% RSLogix 500 project I2P-Hands On 4 - Duncan_Sutton.RSS, saved by version 10.00.00.00 %
PROJECT "UNTITLED"    % processor: Bul.1763 MicroLogix 1100 Series B %

PROGRAM FILES
  LAD 2   15 rungs

DATA FILES
  O0 OUTPUT  4 elements
  I1 INPUT  6 elements
  S2 STATUS  66 elements
  B3 BINARY  1 elements
  T4 TIMER  1 elements
  C5 COUNTER  1 elements
  R6 CONTROL  1 elements
  N7 INTEGER  1 elements
  F8 FLOAT  1 elements

LADDER 2
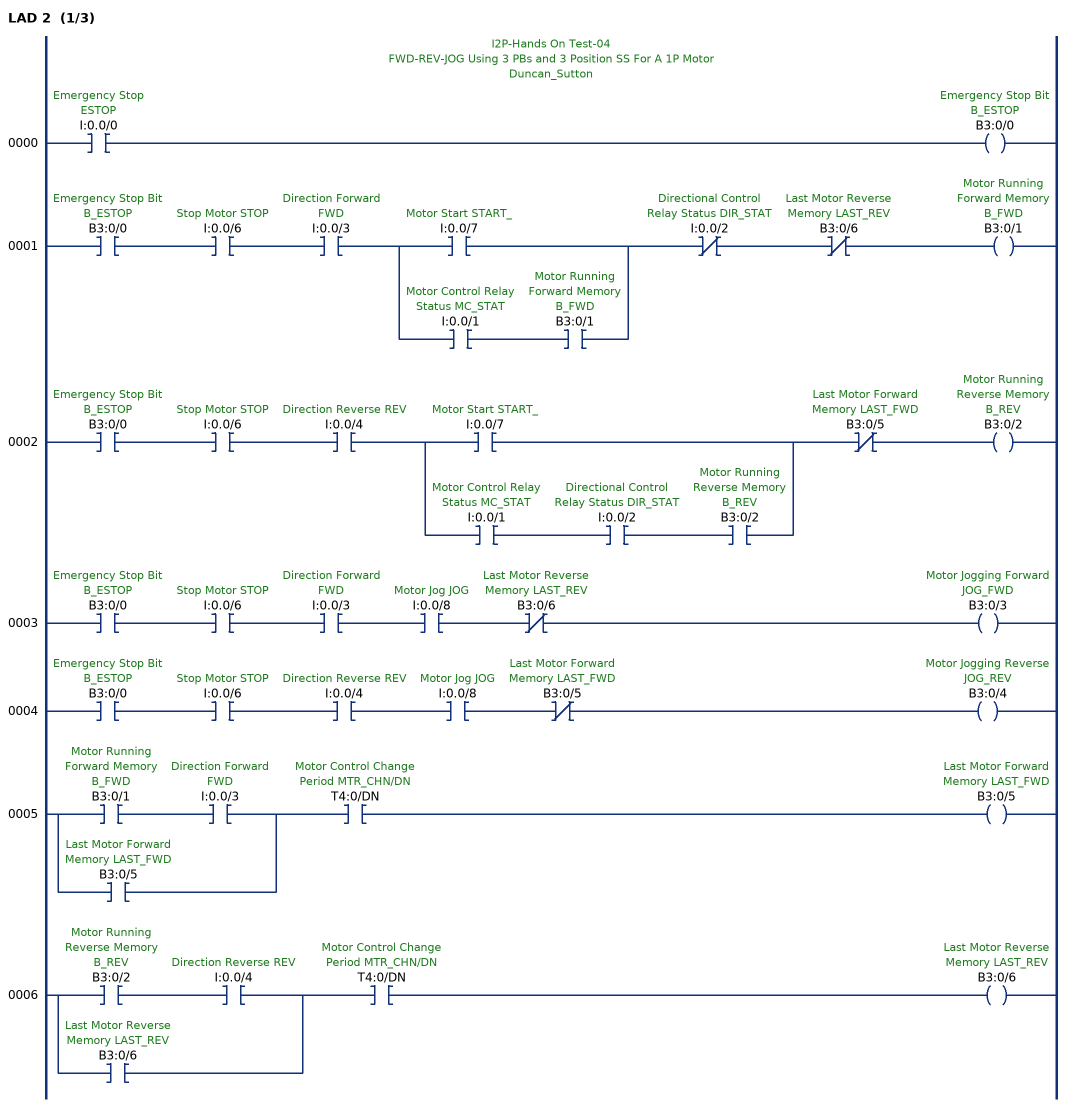
% Rung: 0 %
% I2P-Hands On Test-04
% FWD-REV-JOG Using 3 PBs and 3 Position SS For A 1P Motor
% Duncan_Sutton %
SOR XIC I:0.0/0 OTE B3:0/0 EOR
%   I:0.0/0  ESTOP  "Emergency Stop" %
%   B3:0/0  B_ESTOP  "Emergency Stop Bit" %
% Rung: 1 %
SOR XIC B3:0/0 XIC I:0.0/6 XIC I:0.0/3 BST XIC I:0.0/7 NXB XIC I:0.0/1 XIC B3:0/1 BND XIO I:0.0/2 XIO B3:0/6 OTE B3:0/1 EOR
%   B3:0/0  B_ESTOP  "Emergency Stop Bit" %
%   I:0.0/6  STOP  "Stop Motor" %
%   I:0.0/3  FWD  "Direction Forward" %
%   I:0.0/7  START_  "Motor Start" %
%   I:0.0/1  MC_STAT  "Motor Control Relay Status" %
%   B3:0/1  B_FWD  "Motor Running Forward Memory" %
%   I:0.0/2  DIR_STAT  "Directional Control Relay Status" %
%   B3:0/6  LAST_REV  "Last Motor Reverse Memory" %
% Rung: 2 %
SOR XIC B3:0/0 XIC I:0.0/6 XIC I:0.0/4 BST XIC I:0.0/7 NXB XIC I:0.0/1 XIC I:0.0/2 XIC B3:0/2 BND XIO B3:0/5 OTE B3:0/2 EOR
%   B3:0/0  B_ESTOP  "Emergency Stop Bit" %
%   I:0.0/6  STOP  "Stop Motor" %
%   I:0.0/4  REV  "Direction Reverse" %
%   I:0.0/7  START_  "Motor Start" %
%   I:0.0/1  MC_STAT  "Motor Control Relay Status" %
%   I:0.0/2  DIR_STAT  "Directional Control Relay Status" %
%   B3:0/2  B_REV  "Motor Running Reverse Memory" %
%   B3:0/5  LAST_FWD  "Last Motor Forward Memory" %
% Rung: 3 %
SOR XIC B3:0/0 XIC I:0.0/6 XIC I:0.0/3 XIC I:0.0/8 XIO B3:0/6 OTE B3:0/3 EOR
%   B3:0/0  B_ESTOP  "Emergency Stop Bit" %
%   I:0.0/6  STOP  "Stop Motor" %
%   I:0.0/3  FWD  "Direction Forward" %
%   I:0.0/8  JOG  "Motor Jog" %
%   B3:0/6  LAST_REV  "Last Motor Reverse Memory" %
%   B3:0/3  JOG_FWD  "Motor Jogging Forward" %
% Rung: 4 %
SOR XIC B3:0/0 XIC I:0.0/6 XIC I:0.0/4 XIC I:0.0/8 XIO B3:0/5 OTE B3:0/4 EOR
%   B3:0/0  B_ESTOP  "Emergency Stop Bit" %
%   I:0.0/6  STOP  "Stop Motor" %
%   I:0.0/4  REV  "Direction Reverse" %
%   I:0.0/8  JOG  "Motor Jog" %
%   B3:0/5  LAST_FWD  "Last Motor Forward Memory" %
%   B3:0/4  JOG_REV  "Motor Jogging Reverse" %
% Rung: 5 %
SOR BST XIC B3:0/1 XIC I:0.0/3 NXB XIC B3:0/5 BND XIC T4:0/DN OTE B3:0/5 EOR
%   B3:0/1  B_FWD  "Motor Running Forward Memory" %
%   I:0.0/3  FWD  "Direction Forward" %
%   B3:0/5  LAST_FWD  "Last Motor Forward Memory" %
%   T4:0  MTR_CHN  "Motor Control Change Period" %
% Rung: 6 %
SOR BST XIC B3:0/2 XIC I:0.0/4 NXB XIC B3:0/6 BND XIC T4:0/DN OTE B3:0/6 EOR
%   B3:0/2  B_REV  "Motor Running Reverse Memory" %
%   I:0.0/4  REV  "Direction Reverse" %
%   B3:0/6  LAST_REV  "Last Motor Reverse Memory" %
%   T4:0  MTR_CHN  "Motor Control Change Period" %

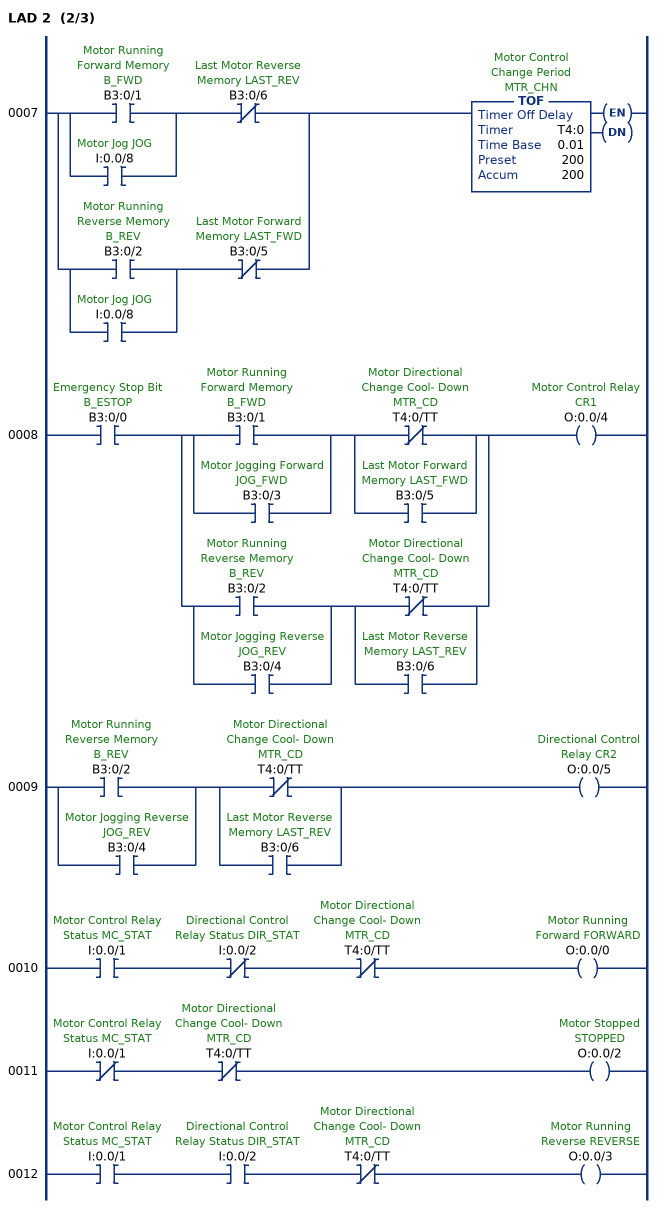
% Rung: 7 %
SOR BST BST XIC B3:0/1 NXB XIC I:0.0/8 BND XIO B3:0/6 NXB BST XIC B3:0/2 NXB XIC I:0.0/8 BND XIO B3:0/5 BND TOF T4:0 0.01 200 200 EOR
%   B3:0/1  B_FWD  "Motor Running Forward Memory" %
%   I:0.0/8  JOG  "Motor Jog" %
%   B3:0/6  LAST_REV  "Last Motor Reverse Memory" %
%   B3:0/2  B_REV  "Motor Running Reverse Memory" %
%   B3:0/5  LAST_FWD  "Last Motor Forward Memory" %
%   T4:0  MTR_CHN  "Motor Control Change Period" %
% Rung: 8 %
SOR XIC B3:0/0 BST BST XIC B3:0/1 NXB XIC B3:0/3 BND BST XIO T4:0/TT NXB XIC B3:0/5 BND NXB BST XIC B3:0/2 NXB XIC B3:0/4 BND BST XIO T4:0/TT NXB XIC B3:0/6 BND BND OTE O:0.0/4 EOR
%   B3:0/0  B_ESTOP  "Emergency Stop Bit" %
%   B3:0/1  B_FWD  "Motor Running Forward Memory" %
%   B3:0/3  JOG_FWD  "Motor Jogging Forward" %
%   T4:0/TT  MTR_CD  "Motor Directional Change Cool- Down" %
%   B3:0/5  LAST_FWD  "Last Motor Forward Memory" %
%   B3:0/2  B_REV  "Motor Running Reverse Memory" %
%   B3:0/4  JOG_REV  "Motor Jogging Reverse" %
%   B3:0/6  LAST_REV  "Last Motor Reverse Memory" %
%   O:0.0/4  CR1  "Motor Control Relay" %
% Rung: 9 %
SOR BST XIC B3:0/2 NXB XIC B3:0/4 BND BST XIO T4:0/TT NXB XIC B3:0/6 BND OTE O:0.0/5 EOR
%   B3:0/2  B_REV  "Motor Running Reverse Memory" %
%   B3:0/4  JOG_REV  "Motor Jogging Reverse" %
%   T4:0/TT  MTR_CD  "Motor Directional Change Cool- Down" %
%   B3:0/6  LAST_REV  "Last Motor Reverse Memory" %
%   O:0.0/5  CR2  "Directional Control Relay" %
% Rung: 10 %
SOR XIC I:0.0/1 XIO I:0.0/2 XIO T4:0/TT OTE O:0.0/0 EOR
%   I:0.0/1  MC_STAT  "Motor Control Relay Status" %
%   I:0.0/2  DIR_STAT  "Directional Control Relay Status" %
%   T4:0/TT  MTR_CD  "Motor Directional Change Cool- Down" %
%   O:0.0/0  FORWARD  "Motor Running Forward" %
% Rung: 11 %
SOR XIO I:0.0/1 XIO T4:0/TT OTE O:0.0/2 EOR
%   I:0.0/1  MC_STAT  "Motor Control Relay Status" %
%   T4:0/TT  MTR_CD  "Motor Directional Change Cool- Down" %
%   O:0.0/2  STOPPED  "Motor Stopped" %
% Rung: 12 %
SOR XIC I:0.0/1 XIC I:0.0/2 XIO T4:0/TT OTE O:0.0/3 EOR
%   I:0.0/1  MC_STAT  "Motor Control Relay Status" %
%   I:0.0/2  DIR_STAT  "Directional Control Relay Status" %
%   T4:0/TT  MTR_CD  "Motor Directional Change Cool- Down" %
%   O:0.0/3  REVERSE  "Motor Running Reverse" %

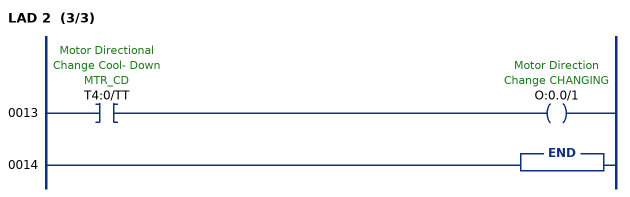
% Rung: 13 %
SOR XIC T4:0/TT OTE O:0.0/1 EOR
%   T4:0/TT  MTR_CD  "Motor Directional Change Cool- Down" %
%   O:0.0/1  CHANGING  "Motor Direction Change" %
% Rung: 14 %
SOR END EOR

OTHER DOCUMENTED ADDRESSES
  START  "Motor Start"

DATA TABLE (non-zero values as saved)
DATA B3
% B3:0 % 0X0001
DATA T4
% .PRE .ACC %
% T4:0 % 200 200
